TYPE ST_InfoDataGroup :
STRUCT
	usiMapState	:USINT;
	usiMapDiag	:USINT;	
END_STRUCT
END_TYPE

(* stored: Version 1.1.0.1, ProductVersion 3.1.4024.12
   DUT ST_InfoDataGroup: Id {e084a955-93d9-4753-b3d6-4a0c307c588b} *)
